// TIA Portal V21 export
VAR_GLOBAL   // PLC tag table "Standard-Variablentabelle"
   "High sensor" AT %I0.0 : Bool;
   "Low sensor" AT %I0.1 : Bool;
   "Pallet sensor" AT %I0.2 : Bool;
   Loaded AT %I0.3 : Bool;
   "At left entry" AT %I0.4 : Bool;
   "At left exit" AT %I0.5 : Bool;
   "At right entry" AT %I0.6 : Bool;
   "At right exit" AT %I0.7 : Bool;
   Start AT %I1.0 : Bool;
   Reset AT %I1.1 : Bool;
   Stop AT %I1.2 : Bool;
   "Emergency stop" AT %I1.3 : Bool;
   Auto AT %I1.4 : Bool;
   Running AT %I1.5 : Bool;
   "Conveyor entry" AT %Q0.0 : Bool;
   Load AT %Q0.1 : Bool;
   Unload AT %Q0.2 : Bool;
   "Trans left" AT %Q0.3 : Bool;
   "Trans right" AT %Q0.4 : Bool;
   "Conveyor left" AT %Q0.5 : Bool;
   "Conveyor right" AT %Q0.6 : Bool;
   "Start light" AT %Q0.7 : Bool;
   "Reset light" AT %Q1.0 : Bool;
   "Stop light" AT %Q1.1 : Bool;
   "Counter" AT %QW30 : Int;
END_VAR
